// TIA Portal V20 export
TYPE "typeSequenceControlNodeHomeCheck"
// stored: Namespace Unit1.Em10
   STRUCT
      liftDownCoverUpPartNoDetect : Bool;
      liftDownCoverUpPartDetect : Bool;
      liftDownCoverDownPartDetect : Bool;
      liftUpCoverUp : Bool;
   END_STRUCT;
END_TYPE
